(* IEC 61131-3 sources: iolink/src/types/serialization/Simatic.Ax.IOLink/LittleEndian, 4 files *)

(* ---- BlockDefinition.st ---- *)
// This is generated code. *** DO NOT MODIFY ***

NAMESPACE Simatic.Ax.iolink
FUNCTION SerializeLittle : UDINT
    VAR_INPUT
        offset : UDINT;
    END_VAR
    VAR_IN_OUT
        value : BlockDefinition;
        buffer : ARRAY[*] OF BYTE;
    END_VAR
    SerializeLittle := offset;
    SerializeLittle := System.Serialization.SerializeLittle(offset := SerializeLittle, value := value.BlockNoDefinition, buffer := buffer);
    SerializeLittle := System.Serialization.SerializeLittle(offset := SerializeLittle, value := value.Channel, buffer := buffer);
    SerializeLittle := System.Serialization.SerializeLittle(offset := SerializeLittle, value := value.BlockType, buffer := buffer);
    SerializeLittle := System.Serialization.SerializeLittle(offset := SerializeLittle, value := value.Version, buffer := buffer);
    SerializeLittle := System.Serialization.SerializeLittle(offset := SerializeLittle, value := value.ByteLength, buffer := buffer);
END_FUNCTION

FUNCTION DeserializeLittle : UDINT
    VAR_INPUT
        offset : UDINT;
        buffer : ARRAY[*] OF BYTE;
    END_VAR
    VAR_IN_OUT
        value : BlockDefinition;
    END_VAR
    DeserializeLittle := offset;
    DeserializeLittle := System.Serialization.DeserializeLittle(offset := DeserializeLittle, value := value.BlockNoDefinition, buffer := buffer);
    DeserializeLittle := System.Serialization.DeserializeLittle(offset := DeserializeLittle, value := value.Channel, buffer := buffer);
    DeserializeLittle := System.Serialization.DeserializeLittle(offset := DeserializeLittle, value := value.BlockType, buffer := buffer);
    DeserializeLittle := System.Serialization.DeserializeLittle(offset := DeserializeLittle, value := value.Version, buffer := buffer);
    DeserializeLittle := System.Serialization.DeserializeLittle(offset := DeserializeLittle, value := value.ByteLength, buffer := buffer);
END_FUNCTION
END_NAMESPACE

(* ---- DeviceHeader.st ---- *)
// This is generated code. *** DO NOT MODIFY ***

NAMESPACE Simatic.Ax.iolink
FUNCTION SerializeLittle : UDINT
    VAR_INPUT
        offset : UDINT;
    END_VAR
    VAR_IN_OUT
        value : DeviceHeader;
        buffer : ARRAY[*] OF BYTE;
    END_VAR
    SerializeLittle := offset;
    SerializeLittle := System.Serialization.SerializeLittle(offset := SerializeLittle, value := value.crc32, buffer := buffer);
    SerializeLittle := System.Serialization.SerializeLittle(offset := SerializeLittle, value := value.SourceDestAddress, buffer := buffer);
    SerializeLittle := System.Serialization.SerializeLittle(offset := SerializeLittle, value := value.TypeIdent, buffer := buffer);
    SerializeLittle := System.Serialization.SerializeLittle(offset := SerializeLittle, value := value.ByteLength, buffer := buffer);
    SerializeLittle := System.Serialization.SerializeLittle(offset := SerializeLittle, value := value.NoOfBlocks, buffer := buffer);
END_FUNCTION

FUNCTION DeserializeLittle : UDINT
    VAR_INPUT
        offset : UDINT;
        buffer : ARRAY[*] OF BYTE;
    END_VAR
    VAR_IN_OUT
        value : DeviceHeader;
    END_VAR
    DeserializeLittle := offset;
    DeserializeLittle := System.Serialization.DeserializeLittle(offset := DeserializeLittle, value := value.crc32, buffer := buffer);
    DeserializeLittle := System.Serialization.DeserializeLittle(offset := DeserializeLittle, value := value.SourceDestAddress, buffer := buffer);
    DeserializeLittle := System.Serialization.DeserializeLittle(offset := DeserializeLittle, value := value.TypeIdent, buffer := buffer);
    DeserializeLittle := System.Serialization.DeserializeLittle(offset := DeserializeLittle, value := value.ByteLength, buffer := buffer);
    DeserializeLittle := System.Serialization.DeserializeLittle(offset := DeserializeLittle, value := value.NoOfBlocks, buffer := buffer);
END_FUNCTION
END_NAMESPACE

(* ---- headerType.st ---- *)
// This is generated code. *** DO NOT MODIFY ***

NAMESPACE Simatic.Ax.IOLink
FUNCTION SerializeLittle : UDINT
    VAR_INPUT
        offset : UDINT;
    END_VAR
    VAR_IN_OUT
        value : headerType;
        buffer : ARRAY[*] OF BYTE;
    END_VAR
    SerializeLittle := offset;
    SerializeLittle := Simatic.Ax.IOLink.SerializeLittle(offset := SerializeLittle, value := value.call, buffer := buffer);
    SerializeLittle := Simatic.Ax.IOLink.SerializeLittle(offset := SerializeLittle, value := value.iolHeader, buffer := buffer);
END_FUNCTION

FUNCTION DeserializeLittle : UDINT
    VAR_INPUT
        offset : UDINT;
        buffer : ARRAY[*] OF BYTE;
    END_VAR
    VAR_IN_OUT
        value : headerType;
    END_VAR
    DeserializeLittle := offset;
    DeserializeLittle := Simatic.Ax.IOLink.DeserializeLittle(offset := DeserializeLittle, value := value.call, buffer := buffer);
    DeserializeLittle := Simatic.Ax.IOLink.DeserializeLittle(offset := DeserializeLittle, value := value.iolHeader, buffer := buffer);
END_FUNCTION
END_NAMESPACE

(* ---- statReadWriteType.st ---- *)
// This is generated code. *** DO NOT MODIFY ***

NAMESPACE Simatic.Ax.IOLink
FUNCTION SerializeLittle : UDINT
    VAR_INPUT
        offset : UDINT;
    END_VAR
    VAR_IN_OUT
        value : LIOLink_typeReadWrite;
        buffer : ARRAY[*] OF BYTE;
    END_VAR
    VAR_TEMP
        i : DINT;
    END_VAR
    SerializeLittle := offset;
    SerializeLittle := Simatic.Ax.IOLink.SerializeLittle(offset := SerializeLittle, value := value.header, buffer := buffer);
    FOR i := DINT#0 TO DINT#231 DO
        SerializeLittle := System.Serialization.SerializeLittle(offset := SerializeLittle, value := value.data[i], buffer := buffer);
    END_FOR;
END_FUNCTION

FUNCTION DeserializeLittle : UDINT
    VAR_INPUT
        offset : UDINT;
        buffer : ARRAY[*] OF BYTE;
    END_VAR
    VAR_IN_OUT
        value : LIOLink_typeReadWrite;
    END_VAR
    VAR_TEMP
        i : DINT;
    END_VAR
    DeserializeLittle := offset;
    DeserializeLittle := Simatic.Ax.IOLink.DeserializeLittle(offset := DeserializeLittle, value := value.header, buffer := buffer);
    FOR i := DINT#0 TO DINT#231 DO
        DeserializeLittle := System.Serialization.DeserializeLittle(offset := DeserializeLittle, value := value.data[i], buffer := buffer);
    END_FOR;
END_FUNCTION
END_NAMESPACE
